FUNCTION F_Concat4 : STRING
VAR_INPUT
	s1																	: STRING;
	s2																	: STRING;
	s3																	: STRING;
	s4																	: STRING;
END_VAR
VAR
END_VAR

// F_Concat4
// Rev 1.0 - January 10, 2024

F_Concat4																:= CONCAT(s1, s2);
F_Concat4																:= CONCAT(F_Concat4, s3);
F_Concat4																:= CONCAT(F_Concat4, s4);

END_FUNCTION

(* stored: Version 1.1.0.1, ProductVersion 3.1.4024.12
   POU F_Concat4: Id {31bccea4-9c60-4a6f-9ca7-efa63767e87c}, SpecialFunc None *)
